KUKA KRL data list: $config.dat

&ACCESS RV$
DEFDAT $CONFIG

ENDDAT
